FUNCTION SPLIT_BYTE_INTO_QUARTERS (* this Function extracts the 4 QUARTER BYTE from a byte *)
  (* Standard: 61499-1; Description: Copyright (c) 2024 HR Agrartechnik GmbH This program and the accompanying materials are made available under the terms of the Eclipse Public License 2.0 which is available at https://www.eclipse.org/legal/epl-2.0/ SPDX-License-Identifier: EPL-2.0 *)
  (* Version 1.0, 2024-02-22, Franz H??pfinger, HR Agrartechnik, initial Implementation *)
  (* Version 1.1, 2024-07-24, Moritz Ortmeier, HR Agrartechnik, rename Function and change Output Variables *)
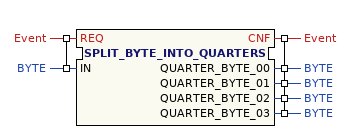
  EVENT_INPUT
    REQ WITH IN;
  END_EVENT
  EVENT_OUTPUT
    CNF WITH QUARTER_BYTE_00, QUARTER_BYTE_01, QUARTER_BYTE_02, QUARTER_BYTE_03;
  END_EVENT
  VAR_INPUT
    IN : BYTE;
  END_VAR
  VAR_OUTPUT
    QUARTER_BYTE_00 : BYTE;
    QUARTER_BYTE_01 : BYTE;
    QUARTER_BYTE_02 : BYTE;
    QUARTER_BYTE_03 : BYTE;
  END_VAR
  BODY IN ST:
(* this Function extracts the 4 QUARTER BYTE from a byte *)
FUNCTION SPLIT_BYTE_INTO_QUARTERS

VAR_INPUT
	IN : BYTE;
END_VAR

VAR_OUTPUT
	QUARTER_BYTE_00 : BYTE;
	QUARTER_BYTE_01 : BYTE;
	QUARTER_BYTE_02 : BYTE;
	QUARTER_BYTE_03 : BYTE;
END_VAR

QUARTER_BYTE_00 := SHR(IN AND quarterconst::BYTE_QUARTER_00, quarterconst::SHIFT_QUARTER_00);
QUARTER_BYTE_01 := SHR(IN AND quarterconst::BYTE_QUARTER_01, quarterconst::SHIFT_QUARTER_01);
QUARTER_BYTE_02 := SHR(IN AND quarterconst::BYTE_QUARTER_02, quarterconst::SHIFT_QUARTER_02);
QUARTER_BYTE_03 := SHR(IN AND quarterconst::BYTE_QUARTER_03, quarterconst::SHIFT_QUARTER_03);

END_FUNCTION
  END_BODY
END_FUNCTION
